{attribute addProperty BoxType "KL6581-0002"}
{attribute addProperty Id "Channel_1Channel_63387A5900"}
{attribute addProperty CRC "4090938439"}
{attribute addProperty SizeInBites "0"}
{attribute addProperty SizeInBytes "0"}
TYPE KL_F3D6C447 :
STRUCT
	{attribute addProperty Name "Channel_1"}
	Channel_1 : Channel_63387A59;
END_STRUCT
END_TYPE

(* stored: Version 1.2.0.0, ProductVersion 3.1.4024.9
   DUT KL_F3D6C447: Id {7cd1bc55-5c75-4ff9-ae38-29c17694e417} *)
